(* PLC project PLC, Beckhoff Automation GmbH TwinCAT PLC Control 3.5.13.21 *)
(* stored: creationDateTime 2023-01-03T15:24:32.5994477, modificationDateTime 2023-01-03T15:24:32.5994477 *)

VAR_GLOBAL  (* GVL_AutoGenerated *)
  EtherCATStatus AT %Q* : UINT;
  EtherCAT_CoEWriteExecute AT %I* : BOOL;
  EtherCAT_CoEWriteError AT %Q* : BOOL;
  EtherCAT_CoEWriteDone AT %Q* : BOOL;
  EtherCAT_CoEWriteSlaveAddr AT %I* : UINT;
  EtherCAT_CoEWriteIndex AT %I* : WORD;
  EtherCAT_CoEWriteSubIndex AT %I* : BYTE;
  EtherCAT_NetId AT %I* : AMSNETID;
  EtherCATChangeCount AT %Q* : ARRAY[1..EtherDeviceCount] OF UINT;
  EtherCATState AT %Q* : ARRAY[1..EtherDeviceCount] OF UINT;
  EtherCATChangeCountReset AT %I* : BOOL;
END_VAR
